{attribute 'qualified_only'}
{attribute 'strict'}
TYPE E_AlarmLevel :
(
	NONE,
	INFO,
	WARNING,
	ERROR
);
END_TYPE

(* stored: Version 1.1.0.1, ProductVersion 3.1.4024.13
   DUT E_AlarmLevel: Id {ea2b4f07-b286-0f39-3b58-48802d660b08} *)
